TYPE ST_BigBagActualMassStoreInValues :
STRUCT
    bBigBagChangeHandlerDone : BOOL; // zakończona inicjalizacja nowego worka
    rBagInitialMass          : REAL; // masa początkowa nowego worka

    bMassBalanceDone         : BOOL; // zakończony bilans masy worka po cyklu
    bBagChangeRequired       : BOOL; // bilans wykazał konieczność wymiany worka
    rBagActualMassNew        : REAL; // masa worka po aktualnym cyklu
END_STRUCT
END_TYPE

(* stored: Version 1.1.0.1, ProductVersion 3.1.4024.16
   DUT ST_BigBagActualMassStoreInValues: Id {f970537c-a278-40cc-be46-3f6ffeeb5bc6} *)
